{attribute 'estimated-stack-usage' := '8192'}
// Writes a message, without a tag. The data is length-prefixed.
FUNCTION F_WriteMessage : HRESULT
VAR_IN_OUT
//     fbCtx   : FB_WriteContext;
	stCtx : ST_WriteContext;     
END_VAR
VAR_INPUT
    ipMessage : I_Message;
END_VAR
VAR
    nLength : UDINT;
    aPayload : T_ProtobufRawBuffer;
END_VAR

IF ipMessage = NULL THEN
	F_WriteMessage := F_WriteError(stCtx:= stCtx, eError:= E_WriterErrorCode.InternalError);
	RETURN;
END_IF

F_WriteMessage := ipMessage.Writer.WriteTo(aPayload);
IF FAILED(F_WriteMessage) THEN
	RETURN;
END_IF

nLength := ipMessage.Writer.nBytesWritten;
F_WriteMessage := F_WriteLength(stCtx:= stCtx, nLength:= nLength);
IF FAILED(F_WriteMessage) THEN
	RETURN;
END_IF

F_WriteMessage := F_WriteRawBytes(stCtx:= stCtx, tBytes:= F_ToAnyBytes(aPayload), nLength:= nLength);

END_FUNCTION

(* stored: Version 1.1.0.1
   POU F_WriteMessage: Id {e4751bf1-1312-4dd2-881e-ae3463ea8207}, SpecialFunc None *)
